(* CoDeSys 2.3 export: F_CALC_SENSOR_KG.EXP *)

(* POU FUN/F_CALC_SENSOR_KG, ST *)
FUNCTION F_CALC_SENSOR_KG : BOOL
VAR_INPUT
	IN  : REAL;
END_VAR
VAR_IN_OUT
	Sensor : ST_SENSOR_KG;
END_VAR
VAR
END_VAR
Sensor.Raw := IN * Sensor.Cal_K;
Sensor.Kg  := Sensor.Raw * (Sensor.Cal_C / 100.0);
END_FUNCTION
